// TIA Portal project "PID" (V18)

(* hardware
DEVICE "S7-1200 station_1"  S7-1200 Station
   slot 0: "Rack_0"  S7-1200 Rack  Rack  V1.0
   slot 1: "PLC_1"  CPU 1212C DC/DC/DC  6ES7 212-1AE40-0XB0  V4.6
*)

// ===== PLC "PLC_1"  CPU 1212C DC/DC/DC =====

VAR_GLOBAL   // PLC tag table "Default tag table"
   "Tag_1" AT %Q0.0 : Bool;
   "Tag_2" AT %Q0.0 : Bool;
   "Tag_3" AT %I0.0 : Bool;
   "Tag_4" AT %I0.1 : Bool;
END_VAR

FUNCTION "SET" : Void   // FC1, LAD
{ S7_Optimized_Access := 'TRUE' }
VERSION : 0.1
BEGIN

REGION Network 1
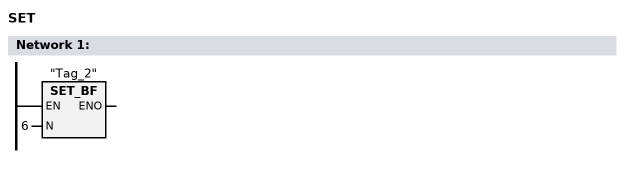
   // no SCL statement known for SBitfield: written as a call
   SET_BF(operand := "Tag_2", n := 6);
END_REGION
END_FUNCTION

FUNCTION "RESET" : Void   // FC2, LAD
{ S7_Optimized_Access := 'TRUE' }
VERSION : 0.1
BEGIN

REGION Network 1
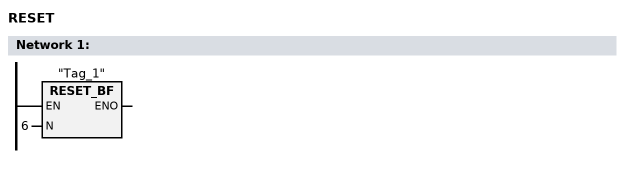
   // no SCL statement known for RBitfield: written as a call
   RESET_BF(operand := "Tag_1", n := 6);
END_REGION
END_FUNCTION

ORGANIZATION_BLOCK "Main"   // OB1, LAD, ProgramCycle
TITLE = "Main Program Sweep (Cycle)"
{ S7_Optimized_Access := 'TRUE' }
VERSION : 0.1
   VAR_INPUT
      Initial_Call : Bool;   // Initial call of this OB
      Remanence : Bool;   // =True, if remanent data are available
   END_VAR
BEGIN

REGION Network 1
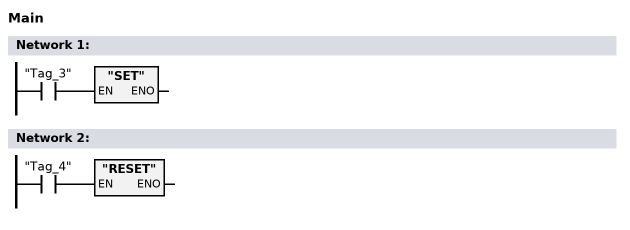
   RUNG wire#powerrail
      Contact( "Tag_3" )
      "SET"()
   END_RUNG
   // the same network as SCL:
   IF "Tag_3" THEN "SET"(); END_IF;
END_REGION

REGION Network 2
   RUNG wire#powerrail
      Contact( "Tag_4" )
      "RESET"()
   END_RUNG
   // the same network as SCL:
   IF "Tag_4" THEN "RESET"(); END_IF;
END_REGION
END_ORGANIZATION_BLOCK